% RSLogix 500 project tripper_GaryS_fixed.RSS, saved by version 8.30.00.16 %
PROJECT "UNTITLED"    % processor: Bul.1763 MicroLogix 1100 Series B %

PROGRAM FILES
  LAD 2   8 rungs
  LAD 3 "SIMULATOR"  11 rungs  % Simulator %

DATA FILES
  O0 OUTPUT  4 elements
  I1 INPUT  6 elements
  S2 STATUS  66 elements
  B3 BINARY  1 elements
  T4 TIMER  1 elements
  C5 COUNTER  1 elements
  R6 CONTROL  1 elements
  N7 INTEGER  4 elements
  F8 FLOAT  1 elements
  N100 SIMUL_INTS  50 elements

LADDER 2
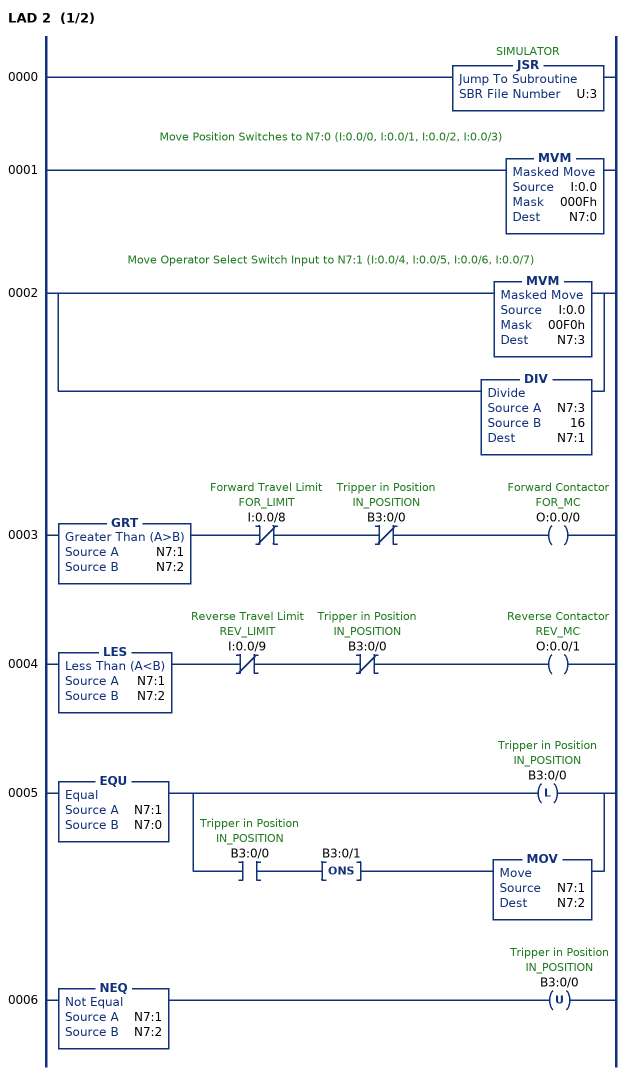
% Rung: 0 %
SOR JSR U:3 EOR
%   U:3  SIMULATOR %
% Rung: 1 %
% Move Position Switches to N7:0 (I:0.0/0, I:0.0/1, I:0.0/2, I:0.0/3) %
SOR MVM I:0.0 000Fh N7:0 EOR
% Rung: 2 %
% Move Operator Select Switch Input to N7:1 (I:0.0/4, I:0.0/5, I:0.0/6, I:0.0/7) %
SOR BST MVM I:0.0 00F0h N7:3 NXB DIV N7:3 16 N7:1 BND EOR
% Rung: 3 %
SOR GRT N7:1 N7:2 XIO I:0.0/8 XIO B3:0/0 OTE O:0.0/0 EOR
%   I:0.0/8  FOR_LIMIT  "Forward Travel Limit" %
%   B3:0/0  IN_POSITION  "Tripper in Position" %
%   O:0.0/0  FOR_MC  "Forward Contactor" %
% Rung: 4 %
SOR LES N7:1 N7:2 XIO I:0.0/9 XIO B3:0/0 OTE O:0.0/1 EOR
%   I:0.0/9  REV_LIMIT  "Reverse Travel Limit" %
%   B3:0/0  IN_POSITION  "Tripper in Position" %
%   O:0.0/1  REV_MC  "Reverse Contactor" %
% Rung: 5 %
SOR EQU N7:1 N7:0 BST OTL B3:0/0 NXB XIC B3:0/0 ONS B3:0/1 MOV N7:1 N7:2 BND EOR
%   B3:0/0  IN_POSITION  "Tripper in Position" %
% Rung: 6 %
SOR NEQ N7:1 N7:2 OTU B3:0/0 EOR
%   B3:0/0  IN_POSITION  "Tripper in Position" %

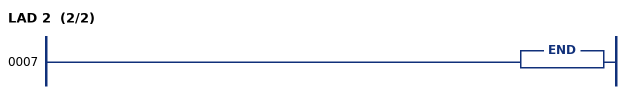
% Rung: 7 %
SOR END EOR

LADDER 3 "SIMULATOR"    % Simulator %
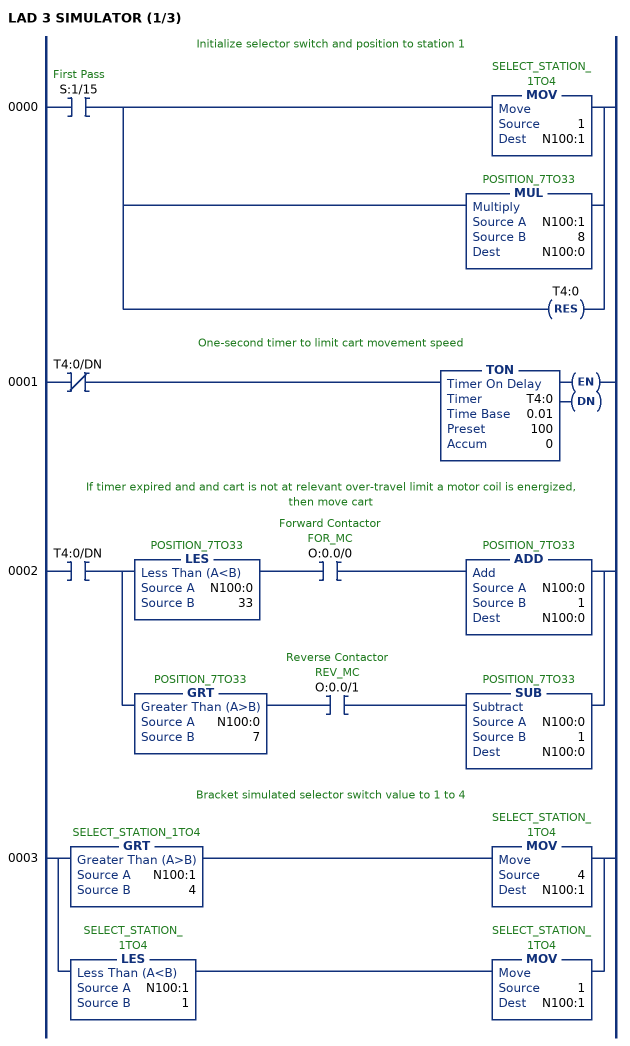
% Rung: 0 %
% Initialize selector switch and position to station 1 %
SOR XIC S:1/15 BST MOV 1 N100:1 NXB MUL N100:1 8 N100:0 NXB RES T4:0 BND EOR
%   S:1/15  "First Pass" %
%   N100:1  SELECT_STATION_1TO4 %
%   N100:0  POSITION_7TO33 %
% Rung: 1 %
% One-second timer to limit cart movement speed %
SOR XIO T4:0/DN TON T4:0 0.01 100 0 EOR
% Rung: 2 %
% If timer expired and and cart is not at relevant over-travel limit a motor coil is energized, then move cart %
SOR XIC T4:0/DN BST LES N100:0 33 XIC O:0.0/0 ADD N100:0 1 N100:0 NXB GRT N100:0 7 XIC O:0.0/1 SUB N100:0 1 N100:0 BND EOR
%   N100:0  POSITION_7TO33 %
%   O:0.0/0  FOR_MC  "Forward Contactor" %
%   O:0.0/1  REV_MC  "Reverse Contactor" %
% Rung: 3 %
% Bracket simulated selector switch value to 1 to 4 %
SOR BST GRT N100:1 4 MOV 4 N100:1 NXB LES N100:1 1 MOV 1 N100:1 BND EOR
%   N100:1  SELECT_STATION_1TO4 %

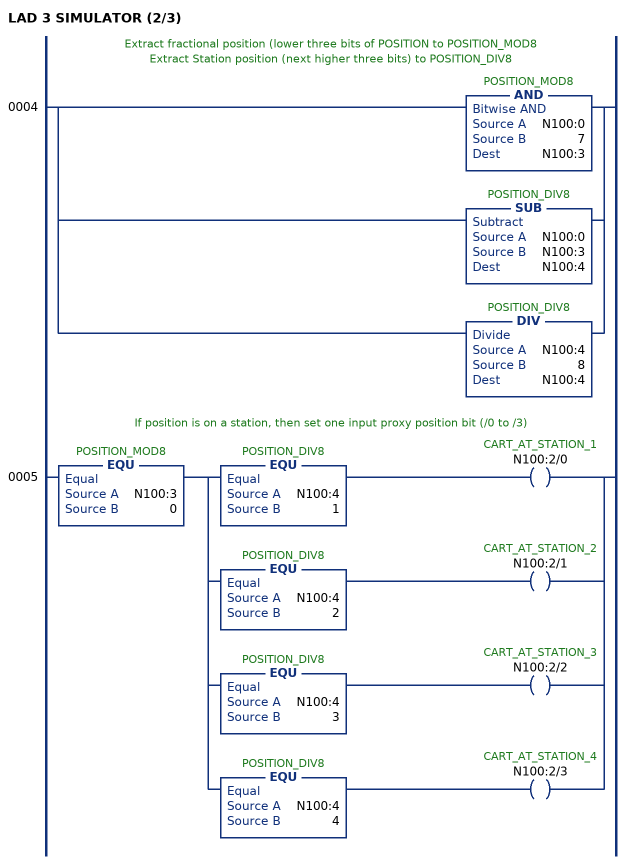
% Rung: 4 %
% Extract fractional position (lower three bits of POSITION to POSITION_MOD8
% Extract Station position (next higher three bits) to POSITION_DIV8 %
SOR BST AND N100:0 7 N100:3 NXB SUB N100:0 N100:3 N100:4 NXB DIV N100:4 8 N100:4 BND EOR
%   N100:0  POSITION_7TO33 %
%   N100:3  POSITION_MOD8 %
%   N100:4  POSITION_DIV8 %
% Rung: 5 %
% If position is on a station, then set one input proxy position bit (/0 to /3) %
SOR EQU N100:3 0 BST EQU N100:4 1 OTE N100:2/0 NXB EQU N100:4 2 OTE N100:2/1 NXB EQU N100:4 3 OTE N100:2/2 NXB EQU N100:4 4 OTE N100:2/3 BND EOR
%   N100:3  POSITION_MOD8 %
%   N100:4  POSITION_DIV8 %
%   N100:2/0  CART_AT_STATION_1 %
%   N100:2/1  CART_AT_STATION_2 %
%   N100:2/2  CART_AT_STATION_3 %
%   N100:2/3  CART_AT_STATION_4 %

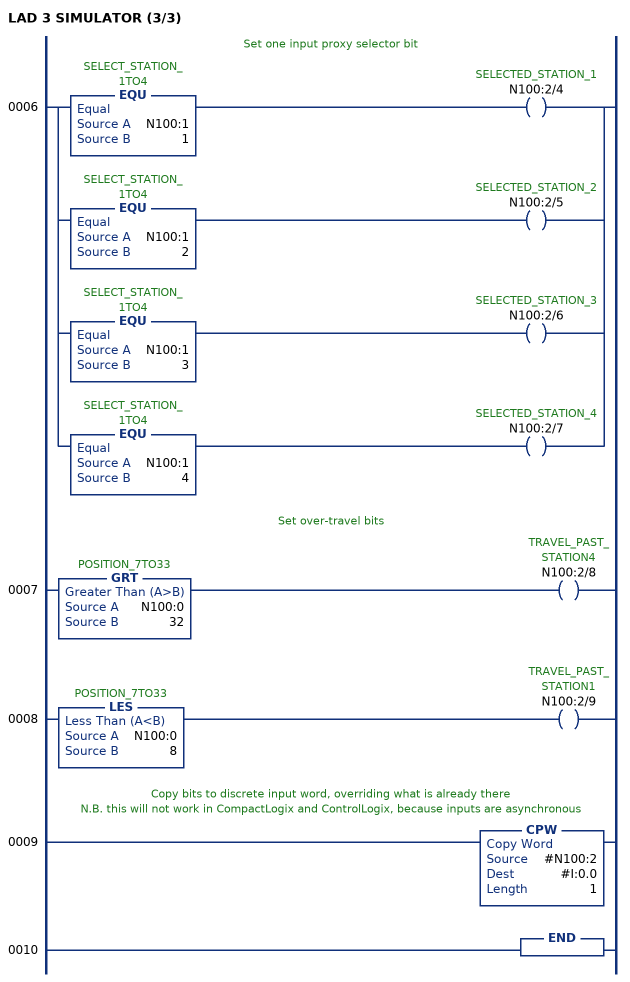
% Rung: 6 %
% Set one input proxy selector bit %
SOR BST EQU N100:1 1 OTE N100:2/4 NXB EQU N100:1 2 OTE N100:2/5 NXB EQU N100:1 3 OTE N100:2/6 NXB EQU N100:1 4 OTE N100:2/7 BND EOR
%   N100:1  SELECT_STATION_1TO4 %
%   N100:2/4  SELECTED_STATION_1 %
%   N100:2/5  SELECTED_STATION_2 %
%   N100:2/6  SELECTED_STATION_3 %
%   N100:2/7  SELECTED_STATION_4 %
% Rung: 7 %
% Set over-travel bits %
SOR GRT N100:0 32 OTE N100:2/8 EOR
%   N100:0  POSITION_7TO33 %
%   N100:2/8  TRAVEL_PAST_STATION4 %
% Rung: 8 %
SOR LES N100:0 8 OTE N100:2/9 EOR
%   N100:0  POSITION_7TO33 %
%   N100:2/9  TRAVEL_PAST_STATION1 %
% Rung: 9 %
% Copy bits to discrete input word, overriding what is already there
% N.B. this will not work in CompactLogix and ControlLogix, because inputs are asynchronous %
SOR CPW #N100:2 #I:0.0 1 EOR
%   N100:2  INPUT_PROXY %
% Rung: 10 %
SOR END EOR

DATA TABLE (non-zero values as saved)
DATA T4
% .PRE .ACC %
% T4:0 % 100 0
DATA N100
% N100:0 % 8 1 0 0 0 0 0 0 0 0
